FUNCTION_BLOCK RollerConveyor EXTENDS Conveyor
VAR_INPUT
END_VAR
VAR_OUTPUT
END_VAR
VAR
END_VAR

Super^();

END_FUNCTION_BLOCK

(* stored: Version 1.1.0.1, ProductVersion 3.1.4024.0
   POU RollerConveyor: Id {b1585fb0-7b13-454c-bee3-cef58924ab6e}, SpecialFunc None *)
